// TIA Portal V19 export
FUNCTION "CallManualOperationLines_Unit3" : Void   // FC82, LAD
// stored: SetENOAutomatically false
   VAR_TEMP
      status : Array[0..30] of Word;   // Status of the configuration or line FC
      errorID : Array[0..30] of Word;   // Error ID of the configuration or line FC
      disableUnit3 : Bool;   // Disable control of the Lines
   END_VAR
   VAR CONSTANT
      MECHANIC_NAME_ENABLE : Bool := FALSE;   // Activation of the Mechanic names
   END_VAR
BEGIN

REGION Network 1: Unit 3 Enable Manual Operation
   // Condition to disable manual operation lines in Unit 3
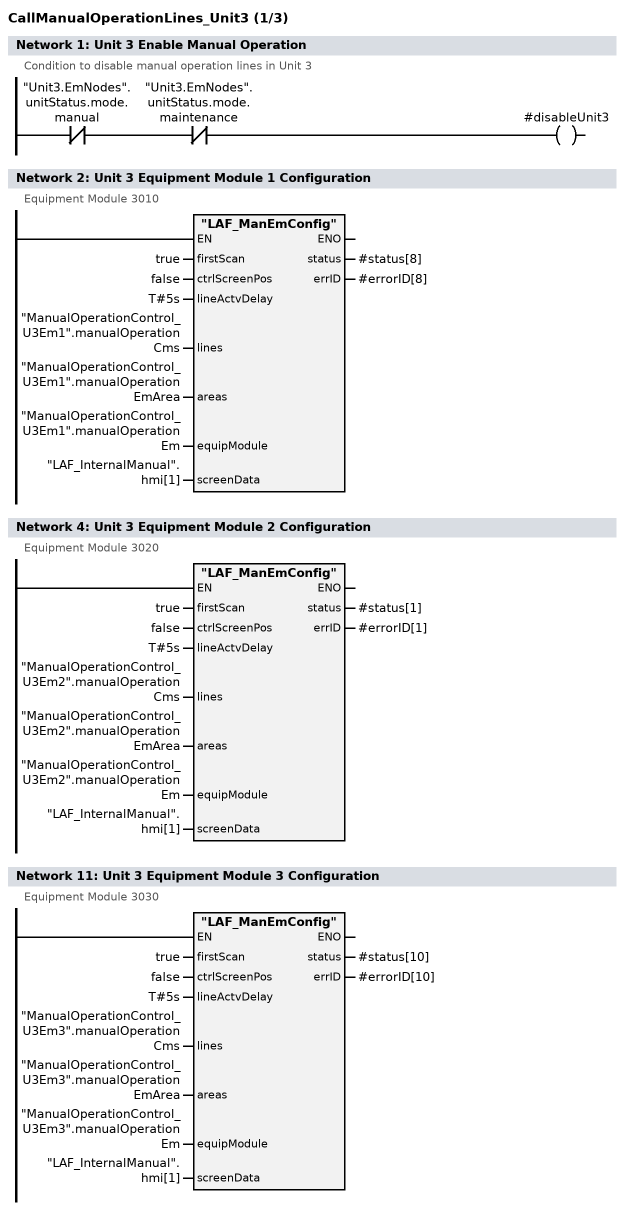
   RUNG wire#powerrail
      I_Contact( "Unit3.EmNodes".unitStatus.mode.manual )
      I_Contact( "Unit3.EmNodes".unitStatus.mode.maintenance )
      Coil( #disableUnit3 )
   END_RUNG
   // the same network as SCL:
   #disableUnit3 := NOT "Unit3.EmNodes".unitStatus.mode.manual AND NOT "Unit3.EmNodes".unitStatus.mode.maintenance;
END_REGION

REGION Network 2: Unit 3 Equipment Module 1 Configuration
   // Equipment Module 3010
   RUNG wire#powerrail
      "LAF_ManEmConfig"(firstScan := true, ctrlScreenPos := false, lineActvDelay := T#5s, lines := "ManualOperationControl_U3Em1".manualOperationCms, areas := "ManualOperationControl_U3Em1".manualOperationEmArea, equipModule := "ManualOperationControl_U3Em1".manualOperationEm, screenData := "LAF_InternalManual".hmi[1], status => #status[8], errID => #errorID[8])
   END_RUNG
   // the same network as SCL:
   "LAF_ManEmConfig"(firstScan := true,
                     ctrlScreenPos := false,
                     lineActvDelay := T#5s,
                     lines := "ManualOperationControl_U3Em1".manualOperationCms,
                     areas := "ManualOperationControl_U3Em1".manualOperationEmArea,
                     equipModule := "ManualOperationControl_U3Em1".manualOperationEm,
                     screenData := "LAF_InternalManual".hmi[1],
                     status => #status[8],
                     errID => #errorID[8]);
END_REGION

REGION Network 3: Unit 3 Equipment Module 1 Line 1
END_REGION

REGION Network 4: Unit 3 Equipment Module 2 Configuration
   // Equipment Module 3020
   RUNG wire#powerrail
      "LAF_ManEmConfig"(firstScan := true, ctrlScreenPos := false, lineActvDelay := T#5s, lines := "ManualOperationControl_U3Em2".manualOperationCms, areas := "ManualOperationControl_U3Em2".manualOperationEmArea, equipModule := "ManualOperationControl_U3Em2".manualOperationEm, screenData := "LAF_InternalManual".hmi[1], status => #status[1], errID => #errorID[1])
   END_RUNG
   // the same network as SCL:
   "LAF_ManEmConfig"(firstScan := true,
                     ctrlScreenPos := false,
                     lineActvDelay := T#5s,
                     lines := "ManualOperationControl_U3Em2".manualOperationCms,
                     areas := "ManualOperationControl_U3Em2".manualOperationEmArea,
                     equipModule := "ManualOperationControl_U3Em2".manualOperationEm,
                     screenData := "LAF_InternalManual".hmi[1],
                     status => #status[1],
                     errID => #errorID[1]);
END_REGION

REGION Network 5: Unit 3 Equipment Module 2 Line 1
   // Line 1 in U3Em2 (Cylinder CM)
END_REGION

REGION Network 6: Unit 3 Equipment Module 2 Line 2
   // Line 2 in U3Em2 (Conveyor CM)
END_REGION

REGION Network 7: Unit 3 Equipment Module 2 Line 3
END_REGION

REGION Network 8: Unit 3 Equipment Module 2 Line 4
END_REGION

REGION Network 9: Unit 3 Equipment Module 2 Line 5
END_REGION

REGION Network 10: Unit 3 Equipment Module 2 Line 6
END_REGION

REGION Network 11: Unit 3 Equipment Module 3 Configuration
   // Equipment Module 3030
   RUNG wire#powerrail
      "LAF_ManEmConfig"(firstScan := true, ctrlScreenPos := false, lineActvDelay := T#5s, lines := "ManualOperationControl_U3Em3".manualOperationCms, areas := "ManualOperationControl_U3Em3".manualOperationEmArea, equipModule := "ManualOperationControl_U3Em3".manualOperationEm, screenData := "LAF_InternalManual".hmi[1], status => #status[10], errID => #errorID[10])
   END_RUNG
   // the same network as SCL:
   "LAF_ManEmConfig"(firstScan := true,
                     ctrlScreenPos := false,
                     lineActvDelay := T#5s,
                     lines := "ManualOperationControl_U3Em3".manualOperationCms,
                     areas := "ManualOperationControl_U3Em3".manualOperationEmArea,
                     equipModule := "ManualOperationControl_U3Em3".manualOperationEm,
                     screenData := "LAF_InternalManual".hmi[1],
                     status => #status[10],
                     errID => #errorID[10]);
END_REGION

REGION Network 12: Unit 3 Equipment Module 3 Line 1
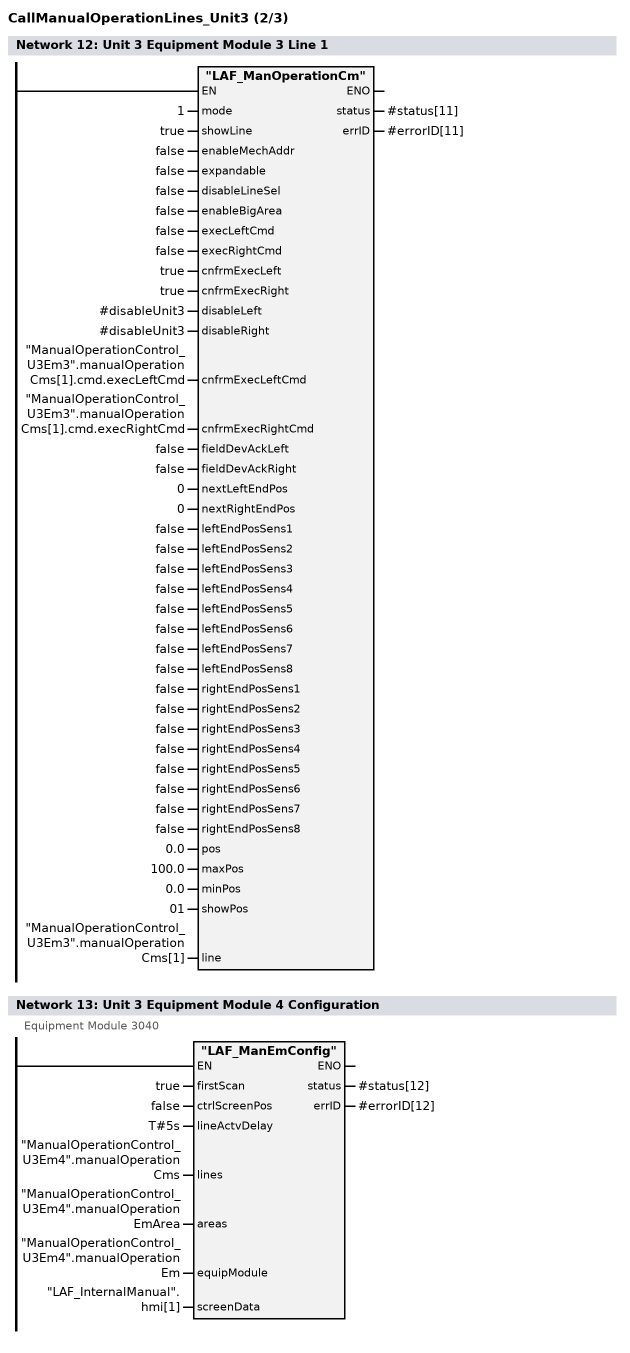
   RUNG wire#powerrail
      "LAF_ManOperationCm"(mode := 1, showLine := true, enableMechAddr := false, expandable := false, disableLineSel := false, enableBigArea := false, execLeftCmd := false, execRightCmd := false, cnfrmExecLeft := true, cnfrmExecRight := true, disableLeft := #disableUnit3, disableRight := #disableUnit3, cnfrmExecLeftCmd := "ManualOperationControl_U3Em3".manualOperationCms[1].cmd.execLeftCmd, cnfrmExecRightCmd := "ManualOperationControl_U3Em3".manualOperationCms[1].cmd.execRightCmd, fieldDevAckLeft := false, fieldDevAckRight := false, nextLeftEndPos := 0, nextRightEndPos := 0, leftEndPosSens1 := false, leftEndPosSens2 := false, leftEndPosSens3 := false, leftEndPosSens4 := false, leftEndPosSens5 := false, leftEndPosSens6 := false, leftEndPosSens7 := false, leftEndPosSens8 := false, rightEndPosSens1 := false, rightEndPosSens2 := false, rightEndPosSens3 := false, rightEndPosSens4 := false, rightEndPosSens5 := false, rightEndPosSens6 := false, rightEndPosSens7 := false, rightEndPosSens8 := false, pos := 0.0, maxPos := 100.0, minPos := 0.0, showPos := 01, line := "ManualOperationControl_U3Em3".manualOperationCms[1], status => #status[11], errID => #errorID[11])
   END_RUNG
   // the same network as SCL:
   "LAF_ManOperationCm"(mode := 1,
                        showLine := true,
                        enableMechAddr := false,
                        expandable := false,
                        disableLineSel := false,
                        enableBigArea := false,
                        execLeftCmd := false,
                        execRightCmd := false,
                        cnfrmExecLeft := true,
                        cnfrmExecRight := true,
                        disableLeft := #disableUnit3,
                        disableRight := #disableUnit3,
                        cnfrmExecLeftCmd := "ManualOperationControl_U3Em3".manualOperationCms[1].cmd.execLeftCmd,
                        cnfrmExecRightCmd := "ManualOperationControl_U3Em3".manualOperationCms[1].cmd.execRightCmd,
                        fieldDevAckLeft := false,
                        fieldDevAckRight := false,
                        nextLeftEndPos := 0,
                        nextRightEndPos := 0,
                        leftEndPosSens1 := false,
                        leftEndPosSens2 := false,
                        leftEndPosSens3 := false,
                        leftEndPosSens4 := false,
                        leftEndPosSens5 := false,
                        leftEndPosSens6 := false,
                        leftEndPosSens7 := false,
                        leftEndPosSens8 := false,
                        rightEndPosSens1 := false,
                        rightEndPosSens2 := false,
                        rightEndPosSens3 := false,
                        rightEndPosSens4 := false,
                        rightEndPosSens5 := false,
                        rightEndPosSens6 := false,
                        rightEndPosSens7 := false,
                        rightEndPosSens8 := false,
                        pos := 0.0,
                        maxPos := 100.0,
                        minPos := 0.0,
                        showPos := 01,
                        line := "ManualOperationControl_U3Em3".manualOperationCms[1],
                        status => #status[11],
                        errID => #errorID[11]);
END_REGION

REGION Network 13: Unit 3 Equipment Module 4 Configuration
   // Equipment Module 3040
   RUNG wire#powerrail
      "LAF_ManEmConfig"(firstScan := true, ctrlScreenPos := false, lineActvDelay := T#5s, lines := "ManualOperationControl_U3Em4".manualOperationCms, areas := "ManualOperationControl_U3Em4".manualOperationEmArea, equipModule := "ManualOperationControl_U3Em4".manualOperationEm, screenData := "LAF_InternalManual".hmi[1], status => #status[12], errID => #errorID[12])
   END_RUNG
   // the same network as SCL:
   "LAF_ManEmConfig"(firstScan := true,
                     ctrlScreenPos := false,
                     lineActvDelay := T#5s,
                     lines := "ManualOperationControl_U3Em4".manualOperationCms,
                     areas := "ManualOperationControl_U3Em4".manualOperationEmArea,
                     equipModule := "ManualOperationControl_U3Em4".manualOperationEm,
                     screenData := "LAF_InternalManual".hmi[1],
                     status => #status[12],
                     errID => #errorID[12]);
END_REGION

REGION Network 14: Unit 3 Equipment Module 4 Line 1
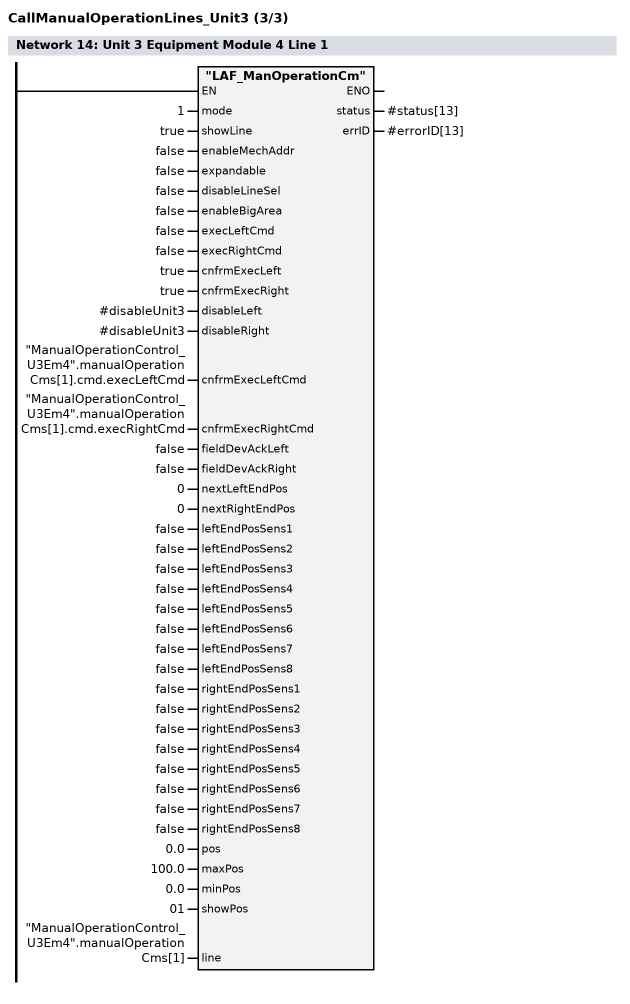
   RUNG wire#powerrail
      "LAF_ManOperationCm"(mode := 1, showLine := true, enableMechAddr := false, expandable := false, disableLineSel := false, enableBigArea := false, execLeftCmd := false, execRightCmd := false, cnfrmExecLeft := true, cnfrmExecRight := true, disableLeft := #disableUnit3, disableRight := #disableUnit3, cnfrmExecLeftCmd := "ManualOperationControl_U3Em4".manualOperationCms[1].cmd.execLeftCmd, cnfrmExecRightCmd := "ManualOperationControl_U3Em4".manualOperationCms[1].cmd.execRightCmd, fieldDevAckLeft := false, fieldDevAckRight := false, nextLeftEndPos := 0, nextRightEndPos := 0, leftEndPosSens1 := false, leftEndPosSens2 := false, leftEndPosSens3 := false, leftEndPosSens4 := false, leftEndPosSens5 := false, leftEndPosSens6 := false, leftEndPosSens7 := false, leftEndPosSens8 := false, rightEndPosSens1 := false, rightEndPosSens2 := false, rightEndPosSens3 := false, rightEndPosSens4 := false, rightEndPosSens5 := false, rightEndPosSens6 := false, rightEndPosSens7 := false, rightEndPosSens8 := false, pos := 0.0, maxPos := 100.0, minPos := 0.0, showPos := 01, line := "ManualOperationControl_U3Em4".manualOperationCms[1], status => #status[13], errID => #errorID[13])
   END_RUNG
   // the same network as SCL:
   "LAF_ManOperationCm"(mode := 1,
                        showLine := true,
                        enableMechAddr := false,
                        expandable := false,
                        disableLineSel := false,
                        enableBigArea := false,
                        execLeftCmd := false,
                        execRightCmd := false,
                        cnfrmExecLeft := true,
                        cnfrmExecRight := true,
                        disableLeft := #disableUnit3,
                        disableRight := #disableUnit3,
                        cnfrmExecLeftCmd := "ManualOperationControl_U3Em4".manualOperationCms[1].cmd.execLeftCmd,
                        cnfrmExecRightCmd := "ManualOperationControl_U3Em4".manualOperationCms[1].cmd.execRightCmd,
                        fieldDevAckLeft := false,
                        fieldDevAckRight := false,
                        nextLeftEndPos := 0,
                        nextRightEndPos := 0,
                        leftEndPosSens1 := false,
                        leftEndPosSens2 := false,
                        leftEndPosSens3 := false,
                        leftEndPosSens4 := false,
                        leftEndPosSens5 := false,
                        leftEndPosSens6 := false,
                        leftEndPosSens7 := false,
                        leftEndPosSens8 := false,
                        rightEndPosSens1 := false,
                        rightEndPosSens2 := false,
                        rightEndPosSens3 := false,
                        rightEndPosSens4 := false,
                        rightEndPosSens5 := false,
                        rightEndPosSens6 := false,
                        rightEndPosSens7 := false,
                        rightEndPosSens8 := false,
                        pos := 0.0,
                        maxPos := 100.0,
                        minPos := 0.0,
                        showPos := 01,
                        line := "ManualOperationControl_U3Em4".manualOperationCms[1],
                        status => #status[13],
                        errID => #errorID[13]);
END_REGION
END_FUNCTION
